{attribute addProperty BoxType "EL3751-0000-0020"}
{attribute addProperty Id "StartTimeNextLatchAT %I*StartTimeNextLatch_356BEDAC648"}
{attribute addProperty CRC "1421024673"}
{attribute addProperty SizeInBites "64"}
{attribute addProperty SizeInBytes "8"}
TYPE PAI_Timestamp_54B31DA1 :
STRUCT
	{attribute addProperty Name "StartTimeNextLatch"}
	StartTimeNextLatch AT %I* : StartTimeNextLatch_356BEDAC;
END_STRUCT
END_TYPE

(* stored: Version 1.2.0.0, ProductVersion 3.1.4024.9
   DUT PAI_Timestamp_54B31DA1: Id {20dfd486-887e-427b-af41-e8c6c8f1b78b} *)
